METHOD PRIVATE RegisterWithDatatypes
VAR_INPUT
END_VAR
IF datatypes = 0 THEN
	RETURN;
END_IF

datatypes.OnEvent('OnDatatypeAdded',THIS^);
END_METHOD

METHOD PROTECTED CreateBundleNode : I_Node
VAR_INPUT
	NodeDatatype : I_StructuredDatatype;
END_VAR
VAR
	pAnyBundleNode : POINTER TO AnyBundleNode;
END_VAR
pAnyBundleNode := __NEW(AnyBundleNode(StructuredDatatype := NodeDatatype));
CreateBundleNode := pAnyBundleNode^;
END_METHOD

METHOD PROTECTED CreateDisplayNode : I_Node
VAR_INPUT
	NodeDatatype : I_Datatype;
END_VAR
VAR
	pAnyDisplayNode : POINTER TO AnyDisplayNode;
END_VAR
pAnyDisplayNode := __NEW(AnyDisplayNode(Datatype := NodeDatatype));
CreateDisplayNode := pAnyDisplayNode^;
END_METHOD

METHOD PROTECTED CreateLiteralNode : I_Node
VAR_INPUT
	NodeDatatype : I_Datatype;
END_VAR
VAR
	pAnyLiteralNode : POINTER TO AnyLiteralNode;
END_VAR
pAnyLiteralNode := __NEW(AnyLiteralNode(Datatype := NodeDatatype));
CreateLiteralNode := pAnyLiteralNode^;
END_METHOD

METHOD PROTECTED CreateUnbundleNode : I_Node
VAR_INPUT
	NodeDatatype : I_StructuredDatatype;
END_VAR
VAR
	pAnyUnbundleNode : POINTER TO AnyUnbundleNode;
END_VAR
pAnyUnbundleNode := __NEW(AnyUnbundleNode(StructuredDatatype := NodeDatatype));
CreateUnbundleNode := pAnyUnbundleNode^;
END_METHOD

METHOD PROTECTED RegisterBundleNodeOfType
VAR_INPUT
	NodeDatatype : I_StructuredDatatype;
END_VAR
VAR
	node : I_Node;
	path : T_MAXSTRING;
END_VAR
node := CreateBundleNode(NodeDatatype);
selfCreatedNodes.Push(node);
path := concat('Bundle/', NodeDatatype.Identifier);
nodeFactory.AddNodeAsPrototype(path,node);
END_METHOD

METHOD PROTECTED RegisterInterfaceDisplayNodeOfType
VAR_INPUT
	NodeDatatype : I_InterfaceDatatype;
END_VAR
VAR
	node : I_Node;
	path : T_MAXSTRING;
END_VAR
node := CreateDisplayNode(NodeDatatype);
selfCreatedNodes.Push(node);
path := concat('Display/', NodeDatatype.Identifier);
nodeFactory.AddNodeAsPrototype(path,node);
END_METHOD

METHOD PROTECTED RegisterInterfaceLiteralNodeOfType
VAR_INPUT
	NodeDatatype : I_InterfaceDatatype;
END_VAR
VAR
	node : I_Node;
	path : T_MAXSTRING;
END_VAR
node := CreateLiteralNode(NodeDatatype);
selfCreatedNodes.Push(node);
path := concat('Literal/', NodeDatatype.Identifier);
nodeFactory.AddNodeAsPrototype(path,node);
END_METHOD

METHOD PROTECTED RegisterPrimitiveDisplayNodeOfType
VAR_INPUT
	NodeDatatype : I_Datatype;
END_VAR
VAR
	node : I_Node;
	path : T_MAXSTRING;
END_VAR
node := CreateDisplayNode(NodeDatatype);
selfCreatedNodes.Push(node);
path := concat('Display/',NodeDatatype.TypeName);
nodeFactory.AddNodeAsPrototype(path,node);
END_METHOD

METHOD PROTECTED RegisterPrimitiveLiteralNodeOfType
VAR_INPUT
	NodeDatatype : I_Datatype;
END_VAR
VAR
	node : I_Node;
	path : T_MAXSTRING;
END_VAR
node := CreateLiteralNode(NodeDatatype);
selfCreatedNodes.Push(node);
path := concat('Literal/',NodeDatatype.TypeName);
nodeFactory.AddNodeAsPrototype(path,node);
END_METHOD

METHOD PROTECTED RegisterUdtDisplayNodeOfType
VAR_INPUT
	NodeDatatype : I_UserDefinedDatatype;
END_VAR
VAR
	node : I_Node;
	path : T_MAXSTRING;
END_VAR
node := CreateDisplayNode(NodeDatatype);
selfCreatedNodes.Push(node);
path := concat('Display/', NodeDatatype.Identifier);
nodeFactory.AddNodeAsPrototype(path,node);
END_METHOD

METHOD PROTECTED RegisterUdtLiteralNodeOfType
VAR_INPUT
	NodeDatatype : I_UserDefinedDatatype;
END_VAR
VAR
	node : I_Node;
	path : T_MAXSTRING;
END_VAR
node := CreateLiteralNode(NodeDatatype);
selfCreatedNodes.Push(node);
path := concat('Literal/', NodeDatatype.Identifier);
nodeFactory.AddNodeAsPrototype(path,node);
END_METHOD

METHOD PROTECTED RegisterUnbundleNodeOfType
VAR_INPUT
	NodeDatatype : I_StructuredDatatype;
END_VAR
VAR
	node : I_Node;
	path : T_MAXSTRING;
END_VAR
node := CreateUnbundleNode(NodeDatatype);
selfCreatedNodes.Push(node);
path := concat('Unbundle/', NodeDatatype.Identifier);
nodeFactory.AddNodeAsPrototype(path,node);
END_METHOD

METHOD PUBLIC HandleEvent
VAR_INPUT
	Event : I_Event;
END_VAR
VAR
	datatypeAddedEvent : I_DatatypeAddedEvent;
	aliasDatatypeAddedEvent : I_AliasDatatypeAddedEvent;
	enumDatatypeAddedEvent : I_EnumDatatypeAddedEvent;
	structuredDatatypeAddedEvent : I_StructuredDatatypeAddedEvent;
	interfaceDatatypeAddedEvent : I_InterfaceDatatypeAddedEvent;
END_VAR
IF __QUERYINTERFACE(event, datatypeAddedEvent) THEN
	RegisterPrimitiveLiteralNodeOfType(datatypeAddedEvent.Target);
	RegisterPrimitiveDisplayNodeOfType(datatypeAddedEvent.Target);
	RETURN;
END_IF

IF __QUERYINTERFACE(event, aliasDatatypeAddedEvent) THEN
	RegisterUdtLiteralNodeOfType(aliasDatatypeAddedEvent.Target);
	RegisterUdtDisplayNodeOfType(aliasDatatypeAddedEvent.Target);
	RETURN;
END_IF

IF __QUERYINTERFACE(event, enumDatatypeAddedEvent) THEN
	RegisterUdtLiteralNodeOfType(enumDatatypeAddedEvent.Target);
	RegisterUdtDisplayNodeOfType(enumDatatypeAddedEvent.Target);
	RETURN;
END_IF

IF __QUERYINTERFACE(event, interfaceDatatypeAddedEvent) THEN
	RegisterInterfaceLiteralNodeOfType(interfaceDatatypeAddedEvent.Target);
	RegisterInterfaceDisplayNodeOfType(interfaceDatatypeAddedEvent.Target);
	RETURN;
END_IF

IF __QUERYINTERFACE(event, structuredDatatypeAddedEvent) THEN
	RegisterUdtLiteralNodeOfType(structuredDatatypeAddedEvent.Target);
	RegisterUdtDisplayNodeOfType(structuredDatatypeAddedEvent.Target);
	RegisterBundleNodeOfType(structuredDatatypeAddedEvent.Target);
	RegisterUnbundleNodeOfType(structuredDatatypeAddedEvent.Target);
	RETURN;
END_IF
END_METHOD

END_FUNCTION_BLOCK

// Node/Bundle/AnyBundleNode
{attribute 'linkalways'} 
{attribute 'no_explicit_call' := 'This FB is a CLASS and must be accessed using methods or properties'}
{attribute 'enable_dynamic_creation'}
FUNCTION_BLOCK FINAL AnyBundleNode EXTENDS Node
VAR
	in : I_StructuredDatatype;
	out : I_StructuredDatatype;
	datatypeOperations : DatatypeOperations;
	selfMadeMembers : Stack;
END_VAR

METHOD FB_init : BOOL
VAR_INPUT
	bInitRetains : BOOL; // if TRUE, the retain variables are initialized (warm start / cold start)
	bInCopyCode : BOOL;  // if TRUE, the instance afterwards gets moved into the copy code (online change)
	StructuredDatatype : I_StructuredDatatype;
END_VAR
VAR
	enumerator : I_KeyValueForwardEnumerator;
	member : I_Datatype;
	memberAsBit : I_BitDatatype;
	memberAsBool : I_Datatype;
	_bool : pointer to _BOOL;
	memberClone : I_Datatype;
END_VAR
StructuredDatatype.Clone().TryResolveAsStructuredDatatype(out);
AddOutput('out', out);

StructuredDatatype.Clone().TryResolveAsStructuredDatatype(in);
enumerator := in.Members.GetMemberEnumerator();

WHILE enumerator.MoveNext() DO 
	IF enumerator.TryGet(member) THEN
		IF member.TryResolveAsBitDatatype(memberAsBit) THEN
			// if the element is a _bit then this needs to be treated differently (as you cannot simply memcpy
			// a bit, as it sits next to other data. Instead, a bool is added in it's place.	
			_bool := __NEW(_BOOL(InitialValue := memberAsBit.Value));
			datatypeOperations.AddWriteBoolToBitOperation(_bool^, memberAsBit);
			AddInput(enumerator.Key, _bool^);
			memberAsBool := _bool^;
			selfMadeMembers.Push(memberAsBool);
		ELSE
			// for all other datatypes,
			memberClone := member.Clone();
			datatypeOperations.AddMemoryCopyOperation(memberClone, member);
			AddInput(enumerator.key, memberClone);
			selfMadeMembers.Push(memberClone);
		END_IF
	END_IF
END_WHILE

enumerator.Dispose();
END_METHOD

METHOD FB_exit : BOOL
VAR_INPUT
	bInCopyCode : BOOL; // if TRUE, the exit method is called for exiting an instance that is copied afterwards (online change).
END_VAR
VAR
	member : I_Datatype;
END_VAR
IF bInCopyCode THEN
	RETURN;
END_IF

in.Dispose();
out.Dispose();
datatypeOperations.Clear();

WHILE selfMadeMembers.TryPop(member) DO
	IF member <> 0 THEN 
		member.dispose();
	END_IF
END_WHILE
END_METHOD

METHOD PUBLIC Clone : I_Node
VAR
	pNode : POINTER TO AnyBundleNode;
END_VAR
pNode := __NEW(AnyBundleNode(StructuredDatatype := in));
Clone := pNode^;
END_METHOD

METHOD PROTECTED OnExecute : HRESULT
VAR
END_VAR
datatypeOperations.Execute();
memcpy(out.Address, in.Address, in.Size);
END_METHOD

END_FUNCTION_BLOCK

// Node/Display/AnyDisplayNode
{attribute 'linkalways'} 
{attribute 'no_explicit_call' := 'This FB is a CLASS and must be accessed using methods or properties'}
{attribute 'enable_dynamic_creation'}
FUNCTION_BLOCK FINAL AnyDisplayNode EXTENDS Node
VAR
	in : I_Datatype;
	display : I_Datatype;
END_VAR

METHOD FB_init : BOOL
VAR_INPUT
	bInitRetains : BOOL; // if TRUE, the retain variables are initialized (warm start / cold start)
	bInCopyCode : BOOL;  // if TRUE, the instance afterwards gets moved into the copy code (online change)
	Datatype : I_Datatype;
END_VAR
THIS^.in := Datatype.Clone();
THIS^.display := Datatype.Clone();

AddInput('in', THIS^.in);
AddContent('display', THIS^.display);
END_METHOD

METHOD FB_exit : BOOL
VAR_INPUT
	bInCopyCode : BOOL; // if TRUE, the exit method is called for exiting an instance that is copied afterwards (online change).
END_VAR
IF bInCopyCode THEN
	RETURN;
END_IF

in.Dispose();
display.Dispose();
END_METHOD

METHOD PUBLIC Clone : I_Node
VAR
	pNode : POINTER TO AnyDisplayNode;
END_VAR
pNode := __NEW(AnyDisplayNode(Datatype := in));
Clone := pNode^;
END_METHOD

METHOD PROTECTED OnExecute : HRESULT
VAR
END_VAR
memcpy(display.Address, in.Address, in.Size);
END_METHOD

END_FUNCTION_BLOCK

// Node/Literal/AnyLiteralNode
{attribute 'linkalways'} 
{attribute 'no_explicit_call' := 'This FB is a CLASS and must be accessed using methods or properties'}
{attribute 'enable_dynamic_creation'}
FUNCTION_BLOCK FINAL AnyLiteralNode EXTENDS Node
VAR
	value : I_Datatype;
	out : I_Datatype;
END_VAR

METHOD FB_init : BOOL
VAR_INPUT
	bInitRetains : BOOL; // if TRUE, the retain variables are initialized (warm start / cold start)
	bInCopyCode : BOOL;  // if TRUE, the instance afterwards gets moved into the copy code (online change)
	Datatype : I_Datatype;
END_VAR
THIS^.value := Datatype.Clone();
THIS^.out := Datatype.Clone();

AddParameter('value', THIS^.value);
AddOutput('out', THIS^.out);
END_METHOD

METHOD FB_exit : BOOL
VAR_INPUT
	bInCopyCode : BOOL; // if TRUE, the exit method is called for exiting an instance that is copied afterwards (online change).
END_VAR
IF bInCopyCode THEN
	RETURN;
END_IF

value.Dispose();
out.Dispose();
END_METHOD

METHOD PUBLIC Clone : I_Node
VAR
	pNode : POINTER TO AnyLiteralNode;
END_VAR
pNode := __NEW(AnyLiteralNode(Datatype := value));
Clone := pNode^;
END_METHOD

METHOD PROTECTED OnExecute : HRESULT
VAR
END_VAR
memcpy(out.Address, value.Address, value.Size);
END_METHOD

END_FUNCTION_BLOCK

// Node/Unbundle/AnyUnbundleNode
{attribute 'linkalways'} 
{attribute 'no_explicit_call' := 'This FB is a CLASS and must be accessed using methods or properties'}
{attribute 'enable_dynamic_creation'}
FUNCTION_BLOCK FINAL AnyUnbundleNode EXTENDS Node
VAR
	in : I_StructuredDatatype;
	out : I_StructuredDatatype;
	datatypeOperations : DatatypeOperations;
	selfMadeMembers : Stack;
END_VAR

METHOD FB_init : BOOL
VAR_INPUT
	bInitRetains : BOOL; // if TRUE, the retain variables are initialized (warm start / cold start)
	bInCopyCode : BOOL;  // if TRUE, the instance afterwards gets moved into the copy code (online change)
	StructuredDatatype : I_StructuredDatatype;
END_VAR
VAR
	enumerator : I_KeyValueForwardEnumerator;
	member : I_Datatype;
	memberAsBit : I_BitDatatype;
	memberAsBool : I_Datatype;
	_bool : Pointer to _BOOL;
	memberClone : I_Datatype;
END_VAR
StructuredDatatype.Clone().TryResolveAsStructuredDatatype(in);
AddInput('in', in);

StructuredDatatype.Clone().TryResolveAsStructuredDatatype(out);
enumerator := out.Members.GetMemberEnumerator();

WHILE enumerator.MoveNext() DO 
	IF enumerator.TryGet(member) THEN
		IF member.TryResolveAsBitDatatype(memberAsBit) THEN
			// if the element is a _bit then this needs to be treated differently (as you cannot simply memcpy
			// a bit, as it sits next to other data. Instead, a bool is added in it's place.	
			_bool := __NEW(_BOOL(InitialValue := memberAsBit.Value));
			datatypeOperations.AddWriteBitToBoolOperation(memberAsBit, _bool^);
			AddOutput(enumerator.Key, _bool^);
			memberAsBool := _bool^;
			selfMadeMembers.Push(memberAsBool);
		ELSE
			// for all other datatypes,
			memberClone := member.Clone();
			datatypeOperations.AddMemoryCopyOperation(member, memberClone);
			AddOutput(enumerator.key, memberClone);
			selfMadeMembers.Push(memberClone);
		END_IF		
	END_IF
END_WHILE

enumerator.Dispose();
END_METHOD

METHOD FB_exit : BOOL
VAR_INPUT
	bInCopyCode : BOOL; // if TRUE, the exit method is called for exiting an instance that is copied afterwards (online change).
END_VAR
VAR
	member : I_Datatype;
END_VAR
IF bInCopyCode THEN
	RETURN;
END_IF

in.Dispose();
out.Dispose();
datatypeOperations.Clear();

WHILE selfMadeMembers.TryPop(member) DO
	IF member <> 0 THEN 
		member.dispose();
	END_IF
END_WHILE
END_METHOD

METHOD PUBLIC Clone : I_Node
VAR
	pNode : POINTER TO AnyUnbundleNode;
END_VAR
pNode := __NEW(AnyUnbundleNode(StructuredDatatype := in));
Clone := pNode^;
END_METHOD

METHOD PROTECTED OnExecute : HRESULT
VAR
END_VAR
memcpy(out.Address, in.Address, in.Size);
datatypeOperations.Execute();
END_METHOD

END_FUNCTION_BLOCK

// Graph/Base/Graph
{attribute 'linkalways'} 
{attribute 'no_explicit_call' := 'This FB is a CLASS and must be accessed using methods or properties'}
{attribute 'enable_dynamic_creation'}
FUNCTION_BLOCK Graph EXTENDS Disposable IMPLEMENTS I_Graph
VAR
	nodeFactory : I_NodeFactory;
	_uuid : T_MAXSTRING;	
	eventEmitter : EventEmitter;
	nodeHost : NodeHost(THIS^, eventEmitter);
	inputPortHost : InputPortHost(THIS^, eventEmitter);
	outputPortHost : OutputPortHost(THIS^, eventEmitter);
	parameterHost : ParameterHost(THIS^, eventEmitter);
	contentHost : ContentHost(THIS^, eventEmitter);
	alarmHost : AlarmHost(THIS^, eventEmitter);
	metadataHost : MetadataHost(THIS^, eventEmitter);
	extensionHost : ExtensionHost(THIS^,eventEmitter);
	selfCreatedNodes : Stack;
	
	deserializationFailedAlarm : DeserializationFailedAlarm(THIS^);
	deserializationFailedNodeNotSupportedAlarm : DeserializationFailedNodeNotSupportedAlarm(THIS^);
END_VAR

METHOD FB_init : BOOL
VAR_INPUT
	bInitRetains : BOOL; // if TRUE, the retain variables are initialized (warm start / cold start)
	bInCopyCode : BOOL;  // if TRUE, the instance afterwards gets moved into the copy code (online change)
	NodeFactory : I_NodeFactory;
END_VAR
THIS^.nodeFactory := NodeFactory;
END_METHOD

METHOD FB_exit : BOOL
VAR_INPUT
	bInCopyCode : BOOL; // if TRUE, the exit method is called for exiting an instance that is copied afterwards (online change).
END_VAR
IF bInCopyCode THEN
	RETURN;
END_IF

DisposeSelfCreatedNodes();
END_METHOD

METHOD PRIVATE DisposeSelfCreatedNodes : BOOL
VAR
	node : I_Node;
END_VAR
WHILE selfCreatedNodes.TryPop(node) DO
	nodeHost.RemoveNode(node);
	node.Dispose();
END_WHILE
END_METHOD

METHOD PUBLIC TryDeserializeLinks : BOOL
VAR_INPUT
	Deserializer : I_Deserializer;
	Feedback : I_DeserializerFeedback;
END_VAR
VAR
	linksDeserializer : I_Deserializer;
	linksEnumerator : I_DeserializerArrayForwardEnumerator;
	linkDeserializer : I_Deserializer;
	sourceNodeId : T_MAXSTRING;
	sourcePortName : T_MAXSTRING;
	destinationNodeId : T_MAXSTRING;
	destinationPortName : T_MAXSTRING;
	sourceNode : I_Node;
	sourcePort : I_OutputPort;
	destinationNode : I_Node;
	destinationPort : I_InputPort;
END_VAR
linksDeserializer := Deserializer.GetKeyArray('links');
linksEnumerator := linksDeserializer.GetArrayEnumerator();

WHILE linksEnumerator.MoveNext() DO
	
	linkDeserializer := linksEnumerator.Current.GetArray();
	
	IF NOT linkDeserializer.GetElementByIndex(1).TryGetString(sourceNodeId, Feedback) THEN
		DeserializationFailedAlarm.Raise('Missing source node id from link');
		linksEnumerator.Dispose();
		RETURN;
	END_IF
	
	IF NOT linkDeserializer.GetElementByIndex(2).TryGetString(sourcePortName, Feedback) THEN
		DeserializationFailedAlarm.Raise('Missing source port name from link');
		linksEnumerator.Dispose();
		RETURN;
	END_IF
	
	IF NOT linkDeserializer.GetElementByIndex(3).TryGetString(destinationNodeId, Feedback) THEN
		DeserializationFailedAlarm.Raise('Missing destination node id from link');
		linksEnumerator.Dispose();
		RETURN;
	END_IF
	
	IF NOT linkDeserializer.GetElementByIndex(4).TryGetString(destinationPortName, Feedback) THEN
		DeserializationFailedAlarm.Raise('Missing destination port name from link');
		linksEnumerator.Dispose();
		RETURN;
	END_IF
	
	IF NOT nodeHost.TryGetNodeById(sourceNodeId, sourceNode) THEN
		DeserializationFailedAlarm.Raise('Unable to get source node when creating link');
		linksEnumerator.Dispose();
		RETURN;
	END_IF
	
	IF NOT nodeHost.TryGetNodeById(destinationNodeId, destinationNode) THEN
		DeserializationFailedAlarm.Raise('Unable to get destination node when creating link');
		linksEnumerator.Dispose();
		RETURN;
	END_IF
	
	IF NOT sourceNode.OutputPorts.TryGetOutputPortByName(sourcePortName, sourcePort) THEN
		DeserializationFailedAlarm.Raise('Unable to get source port when creating link');
		linksEnumerator.Dispose();
		RETURN;
	END_IF
	
	IF NOT destinationNode.InputPorts.TryGetInputPortByName(destinationPortName, destinationPort) THEN
		DeserializationFailedAlarm.Raise('Unable to get destination port when creating link');
		linksEnumerator.Dispose();
		RETURN;
	END_IF
	
	IF NOT destinationPort.TryConnectTo(sourcePort) THEN
		DeserializationFailedAlarm.Raise('Unable to connect source to destination when creating link');
		linksEnumerator.Dispose();
		RETURN;
	END_IF
	
END_WHILE

TryDeserializeLinks := TRUE;
linksEnumerator.Dispose();
END_METHOD

METHOD PUBLIC TryDeserializeNodes : BOOL;
VAR_INPUT
	Deserializer : I_Deserializer;
	Feedback : I_DeserializerFeedback;
END_VAR
VAR
	nodeDeserializer : I_Deserializer;
	nodesEnumerator : I_DeserializerArrayForwardEnumerator;
	nodeType : T_MAXSTRING;
	pError : POINTER TO MissingNodePrototypeDeserializationError;
	node : I_Node;
END_VAR
nodeDeserializer := Deserializer.GetKeyArray('nodes');
nodesEnumerator := nodeDeserializer.GetArrayEnumerator();

WHILE nodesEnumerator.MoveNext() DO
	
	IF NOT nodesEnumerator.Current.TryGetKeyString('type',nodeType, Feedback) THEN
		RETURN;
	END_IF
	
	IF NOT nodeFactory.TryCreateNodeByType(nodeType, node) THEN
		pError := __NEW(MissingNodePrototypeDeserializationError(MissingType := nodeType));
		Feedback.LogError(pError^);
		DeserializationFailedNodeNotSupportedAlarm.Raise(nodeType);
		nodesEnumerator.Dispose();
		RETURN;
	END_IF
	
	selfCreatedNodes.Push(node);
	
	IF NOT node.TryDeserializeFrom(nodesEnumerator.Current, Feedback) THEN
		DeserializationFailedAlarm.Raise('Node failed to deserialize');
		nodesEnumerator.Dispose();
		RETURN;
	END_IF
	
	Nodes.AddNode(node);

END_WHILE

TryDeserializeNodes := TRUE;
nodesEnumerator.Dispose();
END_METHOD

METHOD PUBLIC Accept
VAR_INPUT
	Visitor : I_GraphVisitor;
END_VAR
Visitor.VisitGraph(THIS^);
END_METHOD

METHOD PUBLIC AddMetadata : I_HostMetadata
VAR_INPUT
	Name : T_MAXSTRING;
	Data : I_Datatype;
END_VAR
Metadatum.AddDataAsMetadata(Name, Data);
AddMetadata := THIS^;
END_METHOD

PROPERTY PUBLIC Alarms : I_Alarms
GET
Alarms := alarmHost;
END_GET
END_PROPERTY

PROPERTY PUBLIC Contents : I_Contents
GET
Contents := contentHost;
END_GET
END_PROPERTY

METHOD Execute
VAR_INPUT
END_VAR
nodeHost.Execute();
END_METHOD

PROPERTY PUBLIC Extensions : I_Extensions
GET
Extensions := extensionHost;
END_GET
END_PROPERTY

PROPERTY PUBLIC HasRaisedAlarm : BOOL
GET
HasRaisedAlarm := alarmHost.HasRaisedAlarm;
END_GET
END_PROPERTY

PROPERTY PUBLIC InputPorts : I_InputPorts
GET
InputPorts := inputPortHost;
END_GET
END_PROPERTY

PROPERTY PUBLIC Metadatum : I_Metadatum
GET
Metadatum := metadataHost;
END_GET
END_PROPERTY

PROPERTY PUBLIC Nodes : I_Nodes
GET
Nodes := nodeHost;
END_GET
END_PROPERTY

METHOD PUBLIC OffEvent
VAR_INPUT
	EventName : T_MaxString;
	EventHandler : I_EventHandler;
END_VAR
eventEmitter.OffEvent(EventName, EventHandler);
END_METHOD

METHOD PUBLIC OnceEvent
VAR_INPUT
	EventName : T_MaxString;
	EventHandler : I_EventHandler;
END_VAR
eventEmitter.OnceEvent(EventName, EventHandler);
END_METHOD

METHOD PUBLIC OnEvent
VAR_INPUT
	EventName : T_MaxString;
	EventHandler : I_EventHandler;
END_VAR
eventEmitter.OnEvent(EventName, EventHandler);
END_METHOD

PROPERTY PUBLIC OutputPorts : I_OutputPorts
GET
OutputPorts := outputPortHost;
END_GET
END_PROPERTY

PROPERTY PUBLIC Parameters : I_Parameters
GET
Parameters := parameterHost;
END_GET
END_PROPERTY

METHOD PUBLIC Reset
VAR_INPUT
END_VAR
_uuid := '';
DisposeSelfCreatedNodes();
END_METHOD

METHOD PUBLIC SerializeWith
VAR_INPUT
	Serializer : I_Serializer;
END_VAR
Serializer.StartObject();
Serializer.AddKeyString('uuid',_uuid);
inputPortHost.SerializeWith(Serializer);
outputPortHost.SerializeWith(Serializer);
parameterHost.SerializeWith(Serializer);
contentHost.SerializeWith(Serializer);
alarmHost.SerializeWith(Serializer);
extensionHost.SerializeWith(Serializer);
metadataHost.SerializeWith(Serializer);
nodeHost.SerializeWith(Serializer);
Serializer.EndObject();
END_METHOD

METHOD PUBLIC TryDeserializeFrom : BOOL
VAR_INPUT
	Deserializer : I_Deserializer;
	Feedback : I_DeserializerFeedback;
END_VAR
VAR
	receivedUuid : T_MAXSTRING;
END_VAR
DeserializationFailedNodeNotSupportedAlarm.Clear();
DeserializationFailedAlarm.Clear();

IF NOT parameterHost.TryDeserializeFrom(Deserializer, Feedback) THEN
	RETURN;
END_IF

IF NOT extensionHost.TryDeserializeFrom(Deserializer, Feedback) THEN
	RETURN;
END_IF

IF NOT Deserializer.TryGetKeyString('uuid', receivedUuid, Feedback) THEN
	RETURN;
END_IF

Reset();

IF NOT TryDeserializeNodes(Deserializer, Feedback) THEN 
	RETURN;
END_IF

IF NOT TryDeserializeLinks(Deserializer, Feedback) THEN
	RETURN;
END_IF

_uuid := receivedUuid;
TryDeserializeFrom := TRUE;
END_METHOD

PROPERTY PUBLIC Uuid : T_MAXSTRING
GET
Uuid := _uuid;
END_GET
END_PROPERTY

END_FUNCTION_BLOCK

// Node/Host/NodeHost
{attribute 'linkalways'} 
{attribute 'no_explicit_call' := 'This FB is a CLASS and must be accessed using methods or properties'}
{attribute 'enable_dynamic_creation'}
FUNCTION_BLOCK NodeHost IMPLEMENTS I_Nodes, I_Serializable
VAR
	hostParent : I_HostNodes;
	eventTarget : I_EventTarget;
	nodes : OrderedDictionary;
	nodesInExecutionOrder : LinkedList;
	executeEnumerator : I_ForwardEnumerator;
END_VAR

METHOD FB_init : BOOL
VAR_INPUT
	bInitRetains : BOOL; // if TRUE, the retain variables are initialized (warm start / cold start)
	bInCopyCode : BOOL;  // if TRUE, the instance afterwards gets moved into the copy code (online change)
	Parent : I_HostNodes;
	parentEventTarget : I_EventTarget;
END_VAR
hostParent := Parent;
eventTarget := parentEventTarget;
CreateExecuteEnumerator();
END_METHOD

METHOD FB_exit : BOOL
VAR_INPUT
	bInCopyCode : BOOL; // if TRUE, the exit method is called for exiting an instance that is copied afterwards (online change).
END_VAR
IF bInCopyCode THEN
	RETURN;
END_IF

DestroyExecuteEnumerator();
END_METHOD

METHOD PRIVATE CreateExecuteEnumerator
VAR_INPUT
END_VAR
IF executeEnumerator <> 0 THEN
	executeEnumerator.Dispose();
END_IF

executeEnumerator := nodesInExecutionOrder.GetEnumerator();
END_METHOD

METHOD PRIVATE DestroyExecuteEnumerator
VAR_INPUT
END_VAR
IF executeEnumerator <> 0 THEN
	executeEnumerator.Dispose();
END_IF
END_METHOD

METHOD PROTECTED EmitOnNodeAddedEvent
VAR_INPUT
	Node : I_Node;
END_VAR
VAR
	pNodeAddedEvent : POINTER TO NodeAddedEvent;
END_VAR
IF eventTarget = 0 THEN
	RETURN;
END_IF

pNodeAddedEvent := __NEW(NodeAddedEvent(Target := Node));
eventTarget.Emit('OnNodeAdded',pNodeAddedEvent^);
pNodeAddedEvent^.Dispose();
END_METHOD

METHOD PROTECTED UpdateExecutionOrder
VAR_INPUT
	Node : I_Node;
END_VAR
VAR
	currentPosition : I_LinkedListNode;
	currentNode : I_Node;
END_VAR
// is the list empty?
IF nodesInExecutionOrder.First = 0 THEN
	// if so, add our node first and jump out as done.
	nodesInExecutionOrder.AddFirst(Node);
	RETURN;
END_IF

// if not empty, then is our node higher priorty than the first in the list. 
nodesInExecutionOrder.First.TryGet(currentNode); 
IF currentNode.Order > Node.Order THEN
	// if yes, we are now first, jump out as done. 
	nodesInExecutionOrder.AddFirst(Node);
	RETURN;
END_IF

// here, the list has something in it, and we have less priority than the node in first place.

// get the last node in the list and remember this as "currentPosition" 
currentPosition := nodesInExecutionOrder.Last;

WHILE (TRUE) DO
	
	currentPosition.TryGet(currentNode); 
	// is the current position higer priority than our node?
	IF currentNode.Order <= Node.Order THEN
		// if so, then we go after, jump out as we are done. 
		nodesInExecutionOrder.AddAfter(currentPosition, Node);
		RETURN;
	END_IF
	
	// move one up the list towards the top and try again.
	currentPosition := currentPosition.Previous;

END_WHILE
END_METHOD

METHOD PUBLIC Accept
VAR_INPUT
	Visitor : I_NodeVisitor;
END_VAR
VAR
	enumerator : I_ForwardEnumerator;
	node : I_Node;
END_VAR
enumerator := nodes.GetEnumerator();

WHILE (enumerator.MoveNext()) DO
	
	IF enumerator.TryGet(node) THEN
		node.Accept(Visitor);
	END_IF

END_WHILE

enumerator.Dispose();
END_METHOD

METHOD PUBLIC AddNode
VAR_INPUT
	Node : I_Node;
END_VAR
nodes.AddOrUpdate(Node.id, Node);
UpdateExecutionOrder(Node);
EmitOnNodeAddedEvent(Node);
CreateExecuteEnumerator();
END_METHOD

METHOD PUBLIC Execute
VAR_INPUT
END_VAR
VAR
	node : I_Node;
END_VAR
executeEnumerator.Reset();

WHILE executeEnumerator.MoveNext() DO
	IF executeEnumerator.TryGet(node) THEN
		node.Execute();
	END_IF
END_WHILE
END_METHOD

PROPERTY PUBLIC HasNodes : BOOL
GET
HasNodes := NOT nodes.IsEmpty;
END_GET
END_PROPERTY

METHOD PUBLIC RemoveNode
VAR_INPUT
	Node : I_Node;
END_VAR
nodes.Remove(Node.Id);
nodesInExecutionOrder.Remove(Node);
CreateExecuteEnumerator();
END_METHOD

METHOD PUBLIC SerializeWith
VAR_INPUT
	Serializer : I_Serializer;
END_VAR
VAR
	enumerator : I_ForwardEnumerator;
	node : I_Node;
END_VAR
IF nodes.Count = 0 THEN
	RETURN;
END_IF

Serializer.AddKey('nodes');
Serializer.StartArray();

enumerator := nodes.GetEnumerator();

WHILE enumerator.MoveNext() DO
	IF enumerator.TryGet(node) THEN
		node.SerializeWith(Serializer);
	END_IF
END_WHILE

Serializer.EndArray();
enumerator.Dispose();
END_METHOD

METHOD PUBLIC TryDeserializeFrom : BOOL
VAR_INPUT
	Deserializer : I_Deserializer;
	Feedback : I_DeserializerFeedback;
END_VAR
VAR
	nodeDeserializer : I_Deserializer;
	nodesEnumerator : I_DeserializerArrayForwardEnumerator;
	nodeId : T_MAXSTRING;
	node : I_Node;
END_VAR
nodeDeserializer := Deserializer.GetKeyArray('nodes');
nodesEnumerator := nodeDeserializer.GetArrayEnumerator();

WHILE nodesEnumerator.MoveNext() DO
	
	IF NOT nodesEnumerator.Current.TryGetKeyString('id',nodeId, Feedback) THEN
		CONTINUE;
	END_IF
	
	IF NOT TryGetNodeById(nodeId, node)THEN
		CONTINUE;
	END_IF
	
	node.TryDeserializeFrom(nodesEnumerator.Current, Feedback);

END_WHILE

nodesEnumerator.Dispose();
END_METHOD

METHOD PUBLIC TryGetNodeById : BOOL
VAR_INPUT
	Id : T_MAXSTRING;
	Destination : REFERENCE TO I_Node;
END_VAR
VAR
	node : I_Node;
END_VAR
IF NOT nodes.TryGetValue(Id, node) THEN
	RETURN;
END_IF

Destination := node;
TryGetNodeById := TRUE;
END_METHOD

END_FUNCTION_BLOCK

// Node/Events/NodeAddedEvent
{attribute 'linkalways'} 
{attribute 'no_explicit_call' := 'This FB is a CLASS and must be accessed using methods or properties'}
{attribute 'enable_dynamic_creation'}
FUNCTION_BLOCK NodeAddedEvent EXTENDS Disposable IMPLEMENTS I_NodeAddedEvent
VAR
	_target : I_Node;
END_VAR

METHOD FB_init : BOOL
VAR_INPUT
	bInitRetains : BOOL; // if TRUE, the retain variables are initialized (warm start / cold start)
	bInCopyCode : BOOL;  // if TRUE, the instance afterwards gets moved into the copy code (online change)
	Target : I_Node;
END_VAR
This^._target := Target;
END_METHOD

PROPERTY PUBLIC Target : I_Node
GET
Target := _target;
END_GET
END_PROPERTY

END_FUNCTION_BLOCK

// Node/Events/I_NodeAddedEvent
INTERFACE I_NodeAddedEvent EXTENDS I_Event

PROPERTY PUBLIC Target : I_Node
GET
END_GET
END_PROPERTY

END_INTERFACE

// Errors/MissingNodePrototypeDeserializationError
{attribute 'linkalways'} 
{attribute 'no_explicit_call' := 'This FB is a CLASS and must be accessed using methods or properties'}
{attribute 'enable_dynamic_creation'}
FUNCTION_BLOCK MissingNodePrototypeDeserializationError EXTENDS Error
VAR
	nodeType : T_MAXSTRING;
END_VAR

METHOD FB_init : BOOL
VAR_INPUT
	bInitRetains : BOOL; // if TRUE, the retain variables are initialized (warm start / cold start)
	bInCopyCode : BOOL;  // if TRUE, the instance afterwards gets moved into the copy code (online change)
	MissingType : T_MAXSTRING;
END_VAR
 nodeType := MissingType;
END_METHOD

PROPERTY PUBLIC ErrorType : T_MAXSTRING
GET
ErrorType := 'MISSING_NODE_PROTOTYPE_DESERIALIZATION_ERROR';
END_GET
END_PROPERTY

PROPERTY PUBLIC Message : T_MAXSTRING
GET
Message := CONCAT('Deserialization Failed, Missing Node Prototype : ',nodeType);
END_GET
END_PROPERTY

END_FUNCTION_BLOCK

// Graph/Interfaces/I_Graphs
INTERFACE I_Graphs

METHOD PUBLIC Accept
VAR_INPUT
	visitor : I_GraphVisitor;
END_VAR
END_METHOD

METHOD PUBLIC AddGraph
VAR_INPUT
	Graph : I_Graph;
END_VAR
END_METHOD

METHOD PUBLIC DisposeAll
VAR_INPUT
END_VAR
END_METHOD

METHOD PUBLIC Execute
VAR_INPUT
END_VAR
END_METHOD

METHOD PUBLIC RemoveGraph
VAR_INPUT
	Graph : I_Graph;
END_VAR
END_METHOD

METHOD PUBLIC TryGetGraphByUuid : BOOL
VAR_INPUT
	Uuid : T_MAXSTRING;
	Destination : REFERENCE TO I_Graph;
END_VAR
END_METHOD

END_INTERFACE

// API/Visitors/GetStatusVisitor
{attribute 'linkalways'} 
{attribute 'no_explicit_call' := 'This FB is a CLASS and must be accessed using methods or properties'}
{attribute 'enable_dynamic_creation'}
FUNCTION_BLOCK GetStatusVisitor IMPLEMENTS I_GraphVisitor, I_NodeVisitor, I_ExtensionVisitor, I_ContentVisitor, I_AlarmVisitor
VAR
	serializer : I_Serializer;
END_VAR

METHOD PUBLIC Initialize
VAR_INPUT
	Serializer : I_Serializer;
END_VAR
THIS^.serializer := Serializer;
END_METHOD

METHOD VisitAlarm
VAR_INPUT
	VisitingAlarm : I_Alarm;
END_VAR
IF VisitingAlarm.Active THEN
	serializer.StartObject();
	serializer.AddKeyString('message',VisitingAlarm.Message);
	serializer.AddKeyString('reason',VisitingAlarm.Reason);
	serializer.EndObject();
END_IF
END_METHOD

METHOD VisitContent
VAR_INPUT
	VisitingContent : I_Content;
END_VAR
serializer.StartObject();

serializer.AddKeyString('name',VisitingContent.Name);
serializer.AddKeyObject('value',VisitingContent.Data);

serializer.EndObject();
END_METHOD

METHOD VisitExtension
VAR_INPUT
	VisitingExtension : I_Extension;
END_VAR
Serializer.StartObject();
Serializer.AddKeyString('name',VisitingExtension.Name);

IF VisitingExtension.Alarms.HasAlarms THEN
	serializer.addkey('alarms');
	serializer.StartArray();
	VisitingExtension.Alarms.Accept(THIS^);
	serializer.EndArray();
END_IF

IF VisitingExtension.Contents.HasContents THEN
	serializer.addkey('contents');
	serializer.StartArray();
	VisitingExtension.Contents.Accept(THIS^);
	serializer.EndArray();
END_IF

Serializer.EndObject();
END_METHOD

METHOD VisitGraph
VAR_INPUT
	VisitingGraph : I_Graph;
END_VAR
VAR
	includeInGetStatusVisitor : IncludeInGetStatusVisitor;
END_VAR
serializer.StartObject();

serializer.addKeyString('uuid',VisitingGraph.Uuid);

IF VisitingGraph.Alarms.HasRaisedAlarm THEN
	serializer.addkey('alarms');
	serializer.StartArray();
	VisitingGraph.Alarms.Accept(THIS^);
	serializer.EndArray();
END_IF

IF includeInGetStatusVisitor.CheckExtensions(VisitingGraph) THEN
	serializer.addkey('extensions');
	serializer.StartArray();
	VisitingGraph.Extensions.Accept(THIS^);
	serializer.EndArray();
END_IF

IF VisitingGraph.Contents.HasContents THEN
	serializer.addkey('contents');
	serializer.StartArray();
	VisitingGraph.Contents.Accept(THIS^);
	serializer.EndArray();
END_IF

IF VisitingGraph.Nodes.HasNodes THEN
	serializer.addkey('nodes');
	serializer.StartArray();
	VisitingGraph.Nodes.Accept(THIS^);
	serializer.EndArray();
END_IF

serializer.EndObject();
END_METHOD

METHOD VisitNode
VAR_INPUT
	VisitingNode : I_Node;
END_VAR
VAR
	includeInGetStatusVisitor : IncludeInGetStatusVisitor;
END_VAR
IF NOT includeInGetStatusVisitor.CheckNode(VisitingNode) THEN
	RETURN;
END_IF

serializer.StartObject();
serializer.addKeyString('id', VisitingNode.Id);

IF VisitingNode.Alarms.HasRaisedAlarm THEN
	serializer.addkey('alarms');
	serializer.StartArray();
	VisitingNode.Alarms.Accept(THIS^);
	serializer.EndArray();
END_IF

IF includeInGetStatusVisitor.CheckExtensions(VisitingNode) THEN
	serializer.addkey('extensions');
	serializer.StartArray();
	VisitingNode.Extensions.Accept(THIS^);
	serializer.EndArray();
END_IF

IF VisitingNode.Contents.HasContents THEN
	serializer.addkey('contents');
	serializer.StartArray();
	VisitingNode.Contents.Accept(THIS^);
	serializer.EndArray();
END_IF

serializer.EndObject();
END_METHOD

END_FUNCTION_BLOCK

// API/Visitors/IncludeInGetStatusVisitor
{attribute 'linkalways'} 
{attribute 'no_explicit_call' := 'This FB is a CLASS and must be accessed using methods or properties'}
{attribute 'enable_dynamic_creation'}
FUNCTION_BLOCK IncludeInGetStatusVisitor IMPLEMENTS I_NodeVisitor, I_ExtensionVisitor
VAR
	shouldInclude : BOOL;
END_VAR

METHOD PUBLIC CheckExtensions : BOOL;
VAR_INPUT
	ExtensionHost : I_HostExtensions;
END_VAR
shouldInclude := FALSE;
ExtensionHost.Extensions.Accept(THIS^);
CheckExtensions := shouldInclude;
END_METHOD

METHOD PUBLIC CheckNode : BOOL;
VAR_INPUT
	Node : I_Node;
END_VAR
shouldInclude := FALSE;
Node.Accept(THIS^);
CheckNode := shouldInclude;
END_METHOD

METHOD VisitExtension
VAR_INPUT
	VisitingExtension : I_Extension;
END_VAR
IF VisitingExtension.Contents.HasContents THEN
	shouldInclude := TRUE;
	RETURN;
END_IF

IF VisitingExtension.Alarms.HasRaisedAlarm THEN
	shouldInclude := TRUE;
	RETURN;
END_IF
END_METHOD

METHOD VisitNode
VAR_INPUT
	VisitingNode : I_Node;
END_VAR
IF VisitingNode.Contents.HasContents THEN
	shouldInclude := TRUE;
	RETURN;
END_IF

IF VisitingNode.Alarms.HasRaisedAlarm THEN
	shouldInclude := TRUE;
	RETURN;
END_IF

IF VisitingNode.Extensions.HasExtensions THEN
	VisitingNode.Extensions.Accept(THIS^);
END_IF
END_METHOD

END_FUNCTION_BLOCK

// API/Handlers/CreateGraphRpcHandler
{attribute 'linkalways'} 
{attribute 'no_explicit_call' := 'This FB is a CLASS and must be accessed using methods or properties'}
{attribute 'enable_dynamic_creation'}
FUNCTION_BLOCK CreateGraphRpcHandler IMPLEMENTS I_AsynchronousRpcHandler
VAR
	graphFramework : I_GraphFramework;
	graphs : I_Graphs;
	lastGraphUuid : T_MAXSTRING;
END_VAR

METHOD Handle
VAR_INPUT
	Parameters : I_Deserializer;
	Response : I_AsynchronousRpcResponse;
END_VAR
VAR
	graph : I_Graph;
	feedback : DeserializerFeedback;
	graphDeserializer : I_Deserializer;
	serializer : I_Serializer;
	getStatusVisitor : GetStatusVisitor;
END_VAR
IF graphs.TryGetGraphByUuid(lastGraphUuid,graph) THEN
	graphs.RemoveGraph(graph);
	graph.Dispose();
	lastGraphUuid := '';
END_IF

graph := graphFramework.Create();
graphDeserializer := Parameters.GetKeyObject('graph');

IF NOT graph.TryDeserializeFrom(graphDeserializer, feedback) THEN
	Response.RejectWithMessage(feedback.FirstError.Message);
	graph.Dispose();
	RETURN;
END_IF

lastGraphUuid := graph.Uuid;
graphs.AddGraph(graph);

serializer := Response.GetSerializer();
getStatusVisitor.Initialize(serializer);
getStatusVisitor.VisitGraph(graph);
Response.CompleteWithSerializer(serializer);
serializer.Dispose();
END_METHOD

METHOD PUBLIC Initialize
VAR_INPUT
	GraphFramework : I_GraphFramework;
	Graphs : I_Graphs;
END_VAR
THIS^.graphFramework := GraphFramework;
THIS^.graphs := Graphs;
END_METHOD

END_FUNCTION_BLOCK

// API/Handlers/GetBlueprintsRpcHandler
{attribute 'linkalways'} 
{attribute 'no_explicit_call' := 'This FB is a CLASS and must be accessed using methods or properties'}
{attribute 'enable_dynamic_creation'}
FUNCTION_BLOCK GetBlueprintsRpcHandler IMPLEMENTS I_AsynchronousRpcHandler
VAR
	nodeFactory : I_NodeFactory;
END_VAR

METHOD Handle
VAR_INPUT
	Parameters : I_Deserializer;
	Response : I_AsynchronousRpcResponse;
END_VAR
VAR
	visitor : GetBlueprintsVisitor;
	serializer : I_Serializer;
END_VAR
IF nodeFactory = 0 THEN
	Response.RejectWithMessage('GetBlueprintsRpcHandler has not been initialized with a valid nodeFactory object');
	RETURN;
END_IF

serializer := Response.GetSerializer();
visitor.Initialize(serializer);
nodeFactory.Accept(visitor);

Response.CompleteWithSerializer(serializer);
serializer.Dispose();
END_METHOD

METHOD PUBLIC Initialize
VAR_INPUT
	NodeFactory : I_NodeFactory;
END_VAR
this^.nodeFactory := NodeFactory;
END_METHOD

END_FUNCTION_BLOCK

// API/Visitors/GetBlueprintsVisitor
{attribute 'linkalways'} 
{attribute 'no_explicit_call' := 'This FB is a CLASS and must be accessed using methods or properties'}
{attribute 'enable_dynamic_creation'}
FUNCTION_BLOCK GetBlueprintsVisitor IMPLEMENTS I_NodeFactoryVisitor, I_NodePrototypeVisitor, I_NodeVisitor, I_ExtensionVisitor, I_InputPortVisitor, I_OutputPortVisitor, I_MetadataVisitor, I_ContentVisitor, I_ParameterVisitor, I_AlarmVisitor
VAR
	serializer : I_Serializer;
END_VAR

METHOD PUBLIC Initialize
VAR_INPUT
	Serializer : I_Serializer;
END_VAR
THIS^.serializer := Serializer;
END_METHOD

METHOD VisitAlarm
VAR_INPUT
	VisitingAlarm : I_Alarm;
END_VAR
serializer.AddString(VisitingAlarm.Message);
END_METHOD

METHOD VisitContent
VAR_INPUT
	VisitingContent : I_Content;
END_VAR
serializer.StartObject();

serializer.AddKeyString('name',VisitingContent.Name);
serializer.Addkey('datatype');
VisitingContent.Data.SerializeTypeWith(serializer);

IF VisitingContent.Metadatum.HasMetadata THEN
	serializer.addkey('metadata');
	serializer.StartArray();
	VisitingContent.Metadatum.Accept(THIS^);
	serializer.EndArray();
END_IF

serializer.EndObject();
END_METHOD

METHOD VisitExtension
VAR_INPUT
	VisitingExtension : I_Extension;
END_VAR
Serializer.StartObject();
Serializer.AddKeyString('name',VisitingExtension.Name);

IF VisitingExtension.Metadatum.HasMetadata THEN
	serializer.addkey('metadata');
	serializer.StartArray();
	VisitingExtension.Metadatum.Accept(THIS^);
	serializer.EndArray();
END_IF

IF VisitingExtension.Alarms.HasAlarms THEN
	serializer.addkey('alarms');
	serializer.StartArray();
	VisitingExtension.Alarms.Accept(THIS^);
	serializer.EndArray();
END_IF

IF VisitingExtension.InputPorts.HasInputPorts THEN
	serializer.addkey('inputPorts');
	serializer.StartArray();
	VisitingExtension.InputPorts.Accept(THIS^);
	serializer.EndArray();
END_IF

IF VisitingExtension.OutputPorts.HasOutputPorts THEN
	serializer.addkey('outputPorts');
	serializer.StartArray();
	VisitingExtension.OutputPorts.Accept(THIS^);
	serializer.EndArray();
END_IF

IF VisitingExtension.Parameters.HasParameters THEN
	serializer.addkey('parameters');
	serializer.StartArray();
	VisitingExtension.Parameters.Accept(THIS^);
	serializer.EndArray();
END_IF

IF VisitingExtension.Contents.HasContents THEN
	serializer.addkey('contents');
	serializer.StartArray();
	VisitingExtension.Contents.Accept(THIS^);
	serializer.EndArray();
END_IF

Serializer.EndObject();
END_METHOD

METHOD VisitInputPort
VAR_INPUT
	VisitingInputPort : I_InputPort;
END_VAR
serializer.StartObject();

serializer.AddKeyString('name',VisitingInputPort.Name);
serializer.Addkey('datatype');
VisitingInputPort.Data.SerializeTypeWith(serializer);

IF VisitingInputPort.Metadatum.HasMetadata THEN
	serializer.addkey('metadata');
	serializer.StartArray();
	VisitingInputPort.Metadatum.Accept(THIS^);
	serializer.EndArray();
END_IF

serializer.EndObject();
END_METHOD

METHOD VisitMetadatum
VAR_INPUT
	VisitingMetadatum : I_Metadata;
END_VAR
serializer.StartObject();
serializer.AddKeyString('name',VisitingMetadatum.Name);
serializer.AddkeyObject('value',VisitingMetadatum.Data);
serializer.EndObject();
END_METHOD

METHOD VisitNode
VAR_INPUT
	VisitingNode : I_Node;
END_VAR
serializer.StartObject();

IF VisitingNode.Metadatum.HasMetadata THEN
	serializer.addkey('metadata');
	serializer.StartArray();
	VisitingNode.Metadatum.Accept(THIS^);
	serializer.EndArray();
END_IF

IF VisitingNode.Alarms.HasAlarms THEN
	serializer.addkey('alarms');
	serializer.StartArray();
	VisitingNode.Alarms.Accept(THIS^);
	serializer.EndArray();
END_IF

IF VisitingNode.Extensions.HasExtensions THEN
	serializer.addkey('extensions');
	serializer.StartArray();
	VisitingNode.Extensions.Accept(THIS^);
	serializer.EndArray();
END_IF

IF VisitingNode.InputPorts.HasInputPorts THEN
	serializer.addkey('inputPorts');
	serializer.StartArray();
	VisitingNode.InputPorts.Accept(THIS^);
	serializer.EndArray();
END_IF

IF VisitingNode.OutputPorts.HasOutputPorts THEN
	serializer.addkey('outputPorts');
	serializer.StartArray();
	VisitingNode.OutputPorts.Accept(THIS^);
	serializer.EndArray();
END_IF

IF VisitingNode.Parameters.HasParameters THEN
	serializer.addkey('parameters');
	serializer.StartArray();
	VisitingNode.Parameters.Accept(THIS^);
	serializer.EndArray();
END_IF

IF VisitingNode.Contents.HasContents THEN
	serializer.addkey('contents');
	serializer.StartArray();
	VisitingNode.Contents.Accept(THIS^);
	serializer.EndArray();
END_IF

serializer.EndObject();
END_METHOD

METHOD VisitNodeFactory
VAR_INPUT
	VisitingNodeFactory : I_NodeFactory;
END_VAR
serializer.StartObject();
serializer.AddKey('blueprints');
serializer.StartArray();
VisitingNodeFactory.NodePrototypes.Accept(THIS^);
serializer.EndArray();
serializer.EndObject();
END_METHOD

METHOD VisitNodePrototype
VAR_INPUT
	VisitingPrototype : I_NodePrototype;
END_VAR
serializer.StartObject();
serializer.AddKeyString('path',VisitingPrototype.Path);
serializer.AddKey('node');
VisitingPrototype.Node.Accept(THIS^);
serializer.EndObject();
END_METHOD

METHOD VisitOutputPort
VAR_INPUT
	VisitingOutputPort : I_OutputPort;
END_VAR
serializer.StartObject();

serializer.AddKeyString('name',VisitingOutputPort.Name);
serializer.Addkey('datatype');
VisitingOutputPort.Data.SerializeTypeWith(serializer);

IF VisitingOutputPort.Metadatum.HasMetadata THEN
	serializer.addkey('metadata');
	serializer.StartArray();
	VisitingOutputPort.Metadatum.Accept(THIS^);
	serializer.EndArray();
END_IF

serializer.EndObject();
END_METHOD

METHOD VisitParameter
VAR_INPUT
	VisitingProperty : I_Parameter;
END_VAR
serializer.StartObject();

serializer.AddKeyString('name',VisitingProperty.Name);
serializer.Addkey('datatype');
VisitingProperty.Data.SerializeTypeWith(serializer);
serializer.Addkey('defaultValue');
VisitingProperty.Data.SerializeWith(serializer);

IF VisitingProperty.Metadatum.HasMetadata THEN
	serializer.addkey('metadata');
	serializer.StartArray();
	VisitingProperty.Metadatum.Accept(THIS^);
	serializer.EndArray();
END_IF

Serializer.EndObject();
END_METHOD

END_FUNCTION_BLOCK

// API/Handlers/GetContentValueHandler
{attribute 'linkalways'} 
{attribute 'no_explicit_call' := 'This FB is a CLASS and must be accessed using methods or properties'}
{attribute 'enable_dynamic_creation'}
FUNCTION_BLOCK GetContentValueHandler IMPLEMENTS I_AsynchronousRpcHandler
VAR
	graphs : I_Graphs;
END_VAR

METHOD Handle
VAR_INPUT
	Parameters : I_Deserializer;
	Response : I_AsynchronousRpcResponse;
END_VAR
VAR
	graphUuid : T_MAXSTRING;
	nodeId : T_MAXSTRING;
	contentName : T_MAXSTRING;
	visitor : RetrieveNodeContentValue;
	serializer : I_Serializer;
	feedback : DeserializerFeedback;
END_VAR
IF NOT Parameters.TryGetKeyString('graphUuid', graphUuid, feedback) THEN
	Response.RejectWithMessage(feedback.FirstError.Message);
	RETURN;
END_IF

IF NOT Parameters.TryGetKeyString('nodeId', nodeId, feedback) THEN
	Response.RejectWithMessage(feedback.FirstError.Message);
	RETURN;
END_IF

IF NOT Parameters.TryGetKeyString('contentName', contentName, feedback) THEN
	Response.RejectWithMessage(feedback.FirstError.Message);
	RETURN;
END_IF

serializer := Response.GetSerializer();
visitor.Initialize(graphUuid, nodeId, contentName, serializer);
graphs.Accept(visitor);

IF visitor.Error THEN
	Response.RejectWithMessage(visitor.ErrorMessage);
	serializer.Dispose();
	RETURN;
END_IF

IF NOT visitor.Done THEN
	Response.RejectWithMessage('Invalid graphUuid');
	serializer.Dispose();
	RETURN;
END_IF

Response.CompleteWithSerializer(serializer);
serializer.Dispose();
END_METHOD

METHOD PUBLIC Initialize
VAR_INPUT
	Graphs : I_Graphs;
END_VAR
this^.graphs := Graphs;
END_METHOD

END_FUNCTION_BLOCK

// API/Visitors/RetrieveNodeContentValue
{attribute 'linkalways'} 
{attribute 'no_explicit_call' := 'This FB is a CLASS and must be accessed using methods or properties'}
{attribute 'enable_dynamic_creation'}
FUNCTION_BLOCK RetrieveNodeContentValue IMPLEMENTS I_GraphVisitor, I_NodeVisitor, I_ContentVisitor
VAR
	graphUuid : T_MAXSTRING;
	nodeId : T_MAXSTRING;
	contentName : T_MAXSTRING;
	serializer : I_Serializer;
	_done : BOOL;
	_error : BOOL;
	_errorMessage : T_MAXSTRING;
END_VAR

METHOD PRIVATE LogInvalidContentNameError
VAR_INPUT
END_VAR
_errorMessage := 'Invalid Content Name';
_error := TRUE;
END_METHOD

METHOD PRIVATE LogInvalidNodeIdError
VAR_INPUT
END_VAR
_errorMessage := 'Invalid Node Id';
_error := TRUE;
END_METHOD

METHOD PRIVATE Reset
VAR_INPUT
END_VAR
_done := FALSE;
_errorMessage := '';
_error := FALSE;
END_METHOD

PROPERTY PUBLIC Done : BOOL
GET
Done := _done;
END_GET
END_PROPERTY

PROPERTY PUBLIC Error : BOOL
GET
Error := _error;
END_GET
END_PROPERTY

PROPERTY PUBLIC ErrorMessage : T_MAXSTRING
GET
ErrorMessage := _errorMessage;
END_GET
END_PROPERTY

METHOD PUBLIC Initialize
VAR_INPUT
	GraphUuid : T_MAXSTRING;
	NodeId : T_MAXSTRING;
	ContentName : T_MAXSTRING;
	Serializer : I_Serializer;
END_VAR
THIS^.graphUuid := GraphUuid;
THIS^.nodeId := NodeId;
THIS^.contentName := ContentName;
THIS^.serializer := Serializer;
END_METHOD

METHOD VisitContent
VAR_INPUT
	VisitingContent : I_Content;
END_VAR
VisitingContent.SerializeWith(serializer);
END_METHOD

METHOD VisitGraph
VAR_INPUT
	VisitingGraph : I_Graph;
END_VAR
VAR
	node : I_Node;
END_VAR
Reset();

IF NOT (VisitingGraph.Uuid = graphUuid) THEN
	RETURN;
END_IF

IF NOT VisitingGraph.Nodes.TryGetNodeById(nodeId, node) THEN
	LogInvalidNodeIdError();
	RETURN;
END_IF

node.Accept(THIS^);
END_METHOD

METHOD VisitNode
VAR_INPUT
	VisitingNode : I_Node;
END_VAR
VAR
	content : I_Content;
END_VAR
IF NOT VisitingNode.Contents.TryGetContentByName(contentName, content) THEN
	LogInvalidContentNameError();
	RETURN;
END_IF

content.Accept(THIS^);
END_METHOD

END_FUNCTION_BLOCK

// API/Handlers/GetStatusRpcHandler
{attribute 'linkalways'} 
{attribute 'no_explicit_call' := 'This FB is a CLASS and must be accessed using methods or properties'}
{attribute 'enable_dynamic_creation'}
FUNCTION_BLOCK GetStatusRpcHandler IMPLEMENTS I_AsynchronousRpcHandler
VAR
	graphs : I_Graphs;
END_VAR

METHOD Handle
VAR_INPUT
	Parameters : I_Deserializer;
	Response : I_AsynchronousRpcResponse;
END_VAR
VAR
	graphUuid : T_MAXSTRING;
	graph : I_Graph;
	feedback : DeserializerFeedback;
	serializer : I_Serializer;
	getStatusVisitor : GetStatusVisitor;
END_VAR
IF NOT Parameters.TryGetKeyString('graphUuid', graphUuid, feedback) THEN
	Response.RejectWithMessage(feedback.FirstError.Message);
	RETURN;
END_IF

IF NOT graphs.TryGetGraphByUuid(graphUuid,graph) THEN
	Response.RejectWithMessage(concat('Unknown UUID : ',graphUuid));
	RETURN;
END_IF

serializer := Response.GetSerializer();
getStatusVisitor.Initialize(serializer);
getStatusVisitor.VisitGraph(graph);
Response.CompleteWithSerializer(serializer);
serializer.Dispose();
END_METHOD

METHOD PUBLIC Initialize
VAR_INPUT
	Graphs : I_Graphs;
END_VAR
THIS^.graphs := Graphs;
END_METHOD

END_FUNCTION_BLOCK

// API/Handlers/UpdateParameterValueHandler
{attribute 'linkalways'} 
{attribute 'no_explicit_call' := 'This FB is a CLASS and must be accessed using methods or properties'}
{attribute 'enable_dynamic_creation'}
FUNCTION_BLOCK UpdateParameterValueHandler IMPLEMENTS I_AsynchronousRpcHandler
VAR
	graphs : I_Graphs;
END_VAR

METHOD Handle
VAR_INPUT
	Parameters : I_Deserializer;
	Response : I_AsynchronousRpcResponse;
END_VAR
VAR
	graphUuid : T_MAXSTRING;
	graph : I_Graph;
	nodeId : T_MAXSTRING;
	node : I_Node;
	parameterName : T_MAXSTRING;
	parameter : I_Parameter;
	visitor : RetrieveNodeContentValue;
	serializer : I_Serializer;
	feedback : DeserializerFeedback;
END_VAR
IF NOT Parameters.TryGetKeyString('graphUuid', graphUuid, feedback) THEN
	Response.RejectWithMessage(feedback.FirstError.Message);
	RETURN;
END_IF

IF NOT graphs.TryGetGraphByUuid(graphUuid, graph) THEN
	Response.RejectWithMessage('Invalid or missing graphUuid');
	RETURN;
END_IF

IF NOT Parameters.TryGetKeyString('nodeId', nodeId, feedback) THEN
	Response.RejectWithMessage(feedback.FirstError.Message);
	RETURN;
END_IF

IF NOT graph.Nodes.TryGetNodeById(nodeId, node) THEN
	Response.RejectWithMessage('Invalid or missing nodeId');
	RETURN;
END_IF

IF NOT Parameters.TryGetKeyString('parameterName', parameterName, feedback) THEN
	Response.RejectWithMessage(feedback.FirstError.Message);
	RETURN;
END_IF

IF NOT node.Parameters.TryGetParameterByName(parameterName, parameter) THEN
	Response.RejectWithMessage('Invalid or missing parameterName');
	RETURN;
END_IF

IF NOT Parameters.TryDeserializeKeyToObject ('parameterValue', parameter, feedback) THEN
	Response.RejectWithMessage(feedback.FirstError.Message);
	RETURN;
END_IF

Response.CompleteWithString('done');
END_METHOD

METHOD PUBLIC Initialize
VAR_INPUT
	Graphs : I_Graphs;
END_VAR
this^.graphs := Graphs;
END_METHOD

END_FUNCTION_BLOCK

// API/GraphFrameworkApi
{attribute 'linkalways'} 
{attribute 'no_explicit_call' := 'This FB is a CLASS and must be accessed using methods or properties'}
{attribute 'enable_dynamic_creation'}
FUNCTION_BLOCK GraphFrameworkApi IMPLEMENTS I_RpcApi, I_HostGraphs, I_EventEmitter
VAR
	graphFramework : I_GraphFramework;
	eventEmitter : EventEmitter;
	graphHost : GraphHost(THIS^, eventEmitter);
	createGraphRpcHandler : CreateGraphRpcHandler;
	createGraphMultiUserRpcHandler : CreateGraphMultiUserRpcHandler;
	getStatusRpcHandler : GetStatusRpcHandler;
	getBlueprintsRpcHandler : GetBlueprintsRpcHandler;
	getContentValueHandler : GetContentValueHandler;
	updateParameterValueHandler : UpdateParameterValueHandler;
END_VAR

METHOD FB_init : BOOL
VAR_INPUT
	bInitRetains : BOOL; // if TRUE, the retain variables are initialized (warm start / cold start)
	bInCopyCode : BOOL;  // if TRUE, the instance afterwards gets moved into the copy code (online change)
	GraphFramework : I_GraphFramework;
END_VAR
THIS^.graphFramework := GraphFramework;

getBlueprintsRpcHandler.Initialize(GraphFramework.NodeFactory);
getStatusRpcHandler.Initialize(graphHost);
createGraphRpcHandler.Initialize(GraphFramework, graphHost);
createGraphMultiUserRpcHandler.Initialize(GraphFramework, graphHost);
getContentValueHandler.Initialize(graphHost);
updateParameterValueHandler.Initialize(graphHost);
END_METHOD

METHOD FB_exit : BOOL
VAR_INPUT
	bInCopyCode : BOOL; // if TRUE, the exit method is called for exiting an instance that is copied afterwards (online change).
END_VAR
IF bInCopyCode THEN
	RETURN;
END_IF

graphs.DisposeAll();
END_METHOD

METHOD PUBLIC CyclicCall
VAR_INPUT
END_VAR
graphHost.Execute();
END_METHOD

PROPERTY PUBLIC Graphs : I_Graphs
GET
Graphs := graphHost;
END_GET
END_PROPERTY

METHOD PUBLIC OffEvent
VAR_INPUT
	EventName : T_MaxString;
	EventHandler : I_EventHandler;
END_VAR
eventEmitter.OffEvent(EventName, EventHandler);
END_METHOD

METHOD PUBLIC OnceEvent
VAR_INPUT
	EventName : T_MaxString;
	EventHandler : I_EventHandler;
END_VAR
eventEmitter.OnceEvent(EventName, EventHandler);
END_METHOD

METHOD PUBLIC OnEvent
VAR_INPUT
	EventName : T_MaxString;
	EventHandler : I_EventHandler;
END_VAR
eventEmitter.OnEvent(EventName, EventHandler);
END_METHOD

METHOD RegisterAsynchronousRpcHandlersWith
VAR_INPUT
	Host : I_HostAsynchronousRpcHandlers;
END_VAR
Host.RegisterHandler('CreateGraph',createGraphRpcHandler);
Host.RegisterHandler('CreateGraphMultiUser',createGraphMultiUserRpcHandler);
Host.RegisterHandler('GetStatus',getStatusRpcHandler);
Host.RegisterHandler('GetBlueprints',getBlueprintsRpcHandler);
Host.RegisterHandler('GetContentValue',getContentValueHandler);
Host.RegisterHandler('UpdateParameterValue',updateParameterValueHandler);
END_METHOD

METHOD RegisterSynchronousRpcHandlersWith
VAR_INPUT
	Host : I_HostSynchronousRpcHandlers;
END_VAR
// no implementation
END_METHOD

END_FUNCTION_BLOCK

// Graph/Interfaces/I_HostGraphs
INTERFACE I_HostGraphs

PROPERTY Graphs : I_Graphs
GET
END_GET
END_PROPERTY

END_INTERFACE

// Graph/Host/GraphHost
{attribute 'linkalways'} 
{attribute 'no_explicit_call' := 'This FB is a CLASS and must be accessed using methods or properties'}
{attribute 'enable_dynamic_creation'}
FUNCTION_BLOCK GraphHost IMPLEMENTS I_Graphs, I_Serializable
VAR
	hostParent : I_HostGraphs;
	eventTarget : I_EventTarget;
	graphs : OrderedDictionary;	
END_VAR

METHOD FB_init : BOOL
VAR_INPUT
	bInitRetains : BOOL; // if TRUE, the retain variables are initialized (warm start / cold start)
	bInCopyCode : BOOL;  // if TRUE, the instance afterwards gets moved into the copy code (online change)
	Parent : I_HostGraphs;
	ParentEventTarget : I_EventTarget;
END_VAR
hostParent := Parent;
eventTarget := parentEventTarget;
END_METHOD

METHOD PROTECTED EmitOnGraphAddedEvent
VAR_INPUT
	Graph : I_Graph;
END_VAR
VAR
	pGraphAddedEvent : POINTER TO GraphAddedEvent;
END_VAR
IF eventTarget = 0 THEN
	RETURN;
END_IF

pGraphAddedEvent := __NEW(GraphAddedEvent(Target := Graph));
eventTarget.Emit('OnGraphAdded',pGraphAddedEvent^);
pGraphAddedEvent^.Dispose();
END_METHOD

METHOD PUBLIC Accept
VAR_INPUT
	visitor : I_GraphVisitor;
END_VAR
VAR
	enumerator : I_ForwardEnumerator;
	graph : I_Graph;
END_VAR
enumerator := graphs.GetEnumerator();

WHILE (enumerator.MoveNext()) DO
	
	IF enumerator.TryGet(graph) THEN
		graph.Accept(Visitor);
	END_IF

END_WHILE

enumerator.Dispose();
END_METHOD

METHOD PUBLIC AddGraph
VAR_INPUT
	Graph : I_Graph;
END_VAR
graphs.AddOrUpdate(Graph.Uuid, Graph);
EmitOnGraphAddedEvent(Graph);
END_METHOD

METHOD PUBLIC DisposeAll
VAR_INPUT
END_VAR
VAR
	enumerator : I_ForwardEnumerator;
	graph : I_Graph;
END_VAR
enumerator := graphs.GetEnumerator();

WHILE enumerator.MoveNext() DO
	IF enumerator.TryGet(graph) THEN
		graph.Dispose();
	END_IF
END_WHILE

graphs.Clear();

enumerator.Dispose();
END_METHOD

METHOD PUBLIC Execute
VAR_INPUT
END_VAR
VAR
	enumerator : I_ForwardEnumerator;
	graph : I_Graph;
END_VAR
enumerator := graphs.GetEnumerator();

WHILE enumerator.MoveNext() DO
	IF enumerator.TryGet(graph) THEN
		graph.Execute();
	END_IF
END_WHILE

enumerator.Dispose();
END_METHOD

METHOD PUBLIC RemoveGraph
VAR_INPUT
	Graph : I_Graph;
END_VAR
graphs.Remove(Graph.Uuid);
END_METHOD

METHOD PUBLIC SerializeWith
VAR_INPUT
	Serializer : I_Serializer;
END_VAR
VAR
	enumerator : I_ForwardEnumerator;
	graph : I_Graph;
END_VAR
IF graphs.Count = 0 THEN
	RETURN;
END_IF

Serializer.AddKey('graphs');
Serializer.StartArray();

enumerator := graphs.GetEnumerator();

WHILE enumerator.MoveNext() DO
	IF enumerator.TryGet(graph) THEN
		graph.SerializeWith(Serializer);
	END_IF
END_WHILE

Serializer.EndArray();
enumerator.Dispose();
END_METHOD

METHOD PUBLIC TryGetGraphByUuid : BOOL
VAR_INPUT
	Uuid : T_MAXSTRING;
	Destination : REFERENCE TO I_Graph;
END_VAR
VAR
	graph : I_Graph;
END_VAR
IF NOT graphs.TryGetValue(Uuid, graph) THEN
	RETURN;
END_IF

Destination := graph;
TryGetGraphByUuid := TRUE;
END_METHOD

END_FUNCTION_BLOCK

// Graph/Events/GraphAddedEvent
{attribute 'linkalways'} 
{attribute 'no_explicit_call' := 'This FB is a CLASS and must be accessed using methods or properties'}
{attribute 'enable_dynamic_creation'}
FUNCTION_BLOCK GraphAddedEvent EXTENDS Disposable IMPLEMENTS I_GraphAddedEvent
VAR
	_target : I_Graph;
END_VAR

METHOD FB_init : BOOL
VAR_INPUT
	bInitRetains : BOOL; // if TRUE, the retain variables are initialized (warm start / cold start)
	bInCopyCode : BOOL;  // if TRUE, the instance afterwards gets moved into the copy code (online change)
	Target : I_Graph;
END_VAR
This^._target := Target;
END_METHOD

PROPERTY PUBLIC Target : I_Graph
GET
Target := _target;
END_GET
END_PROPERTY

END_FUNCTION_BLOCK

// Graph/Events/I_GraphAddedEvent
INTERFACE I_GraphAddedEvent EXTENDS I_Event

PROPERTY PUBLIC Target : I_Graph
GET
END_GET
END_PROPERTY

END_INTERFACE

// Extensions/Namespace/ExtensionNamespace
{attribute 'linkalways'} 
{attribute 'no_explicit_call' := 'This FB is a CLASS and must be accessed using methods or properties'}
{attribute 'enable_dynamic_creation'}
FUNCTION_BLOCK ExtensionNamespace
VAR
	_extensionName : T_MAXSTRING;
	_targetName : T_MAXSTRING;
	_isExtensionPath : BOOL;
END_VAR

METHOD FB_init : BOOL
VAR_INPUT
	bInitRetains : BOOL; // if TRUE, the retain variables are initialized (warm start / cold start)
	bInCopyCode : BOOL;  // if TRUE, the instance afterwards gets moved into the copy code (online change)
	Path : T_MAXSTRING;
END_VAR
Initialize(Path);
END_METHOD

PROPERTY PUBLIC ExtensionName : T_MAXSTRING
GET
IF NOT _isExtensionPath THEN
	RETURN;
END_IF

ExtensionName := _extensionNAme;
END_GET
END_PROPERTY

METHOD PUBLIC Initialize
VAR_INPUT
	Path : T_MAXSTRING;
END_VAR
_isExtensionPath := FindAndSplitChar(
	sSeparatorChar := '.',  
	pSrcString := ADR(Path),                                  
	pLeftString := ADR(_extensionName),   
	nLeftSize := SIZEOF(_extensionName),                                  
	pRightString := ADR(_targetName), 
	nRightSize := SIZEOF(_targetName),                                
	bSearchFromRight := TRUE 
);
END_METHOD

PROPERTY PUBLIC IsExtensionPath : BOOL
GET
IsExtensionPath := _isExtensionPath;
END_GET
END_PROPERTY

PROPERTY PUBLIC TargetName : T_MAXSTRING
GET
IF NOT _isExtensionPath THEN
	RETURN;
END_IF

TargetName := _targetName;
END_GET
END_PROPERTY

END_FUNCTION_BLOCK

// Extensions/PreExecutionCheck/Alarms/PreExecutionCheckFailedAlarm
{attribute 'linkalways'} 
{attribute 'no_explicit_call' := 'This FB is a CLASS and must be accessed using methods or properties'}
{attribute 'enable_dynamic_creation'}
FUNCTION_BLOCK PUBLIC PreExecutionCheckFailedAlarm EXTENDS Alarm
VAR
	state : (CLEARED, RAISED);
	_reason : T_MAXSTRING;
END_VAR

PROPERTY Active : BOOL
GET
Active := state <> CLEARED;
END_GET
END_PROPERTY

METHOD PUBLIC Clear
_reason := '';
state := CLEARED;
END_METHOD

PROPERTY PUBLIC Message : T_MaxString
GET
Message := 'Pre-execution check failed';
END_GET
END_PROPERTY

METHOD PUBLIC Raise
VAR_INPUT
	Reason : T_MAXSTRING;
END_VAR
_reason := Reason;
state := RAISED;
END_METHOD

PROPERTY Reason : T_MaxString
GET
Reason := _reason;
END_GET
END_PROPERTY

END_FUNCTION_BLOCK

// Extensions/PreExecutionCheck/Checks/I_PreExecutionChecks
INTERFACE I_PreExecutionChecks

METHOD PUBLIC Fail
VAR_INPUT
	Message : T_MAXSTRING;
END_VAR
END_METHOD

PROPERTY PUBLIC Failed : BOOL
GET
END_GET
END_PROPERTY

METHOD PUBLIC IsFalse
VAR_INPUT
	Actual : BOOL;
	Message : T_MAXSTRING;
END_VAR
END_METHOD

METHOD PUBLIC IsTrue
VAR_INPUT
	Actual : BOOL;
	Message : T_MAXSTRING;
END_VAR
END_METHOD

END_INTERFACE

// Extensions/PreExecutionCheck/Checks/PreExecutionChecks
FUNCTION_BLOCK PreExecutionChecks IMPLEMENTS I_PreExecutionChecks
VAR
	hasFailed : BOOL;
	hasFailedReason : T_MAXSTRING;
END_VAR;

METHOD PUBLIC Fail
VAR_INPUT
	Message : T_MAXSTRING;
END_VAR
IF hasFailed THEN
	RETURN;
END_IF

hasFailed := TRUE;
hasFailedReason := Message;
END_METHOD

PROPERTY PUBLIC Failed : BOOL
GET
Failed := hasFailed;
END_GET
END_PROPERTY

METHOD PUBLIC IsFalse
VAR_INPUT
	Actual : BOOL;
	Message : T_MAXSTRING;
END_VAR
IF hasFailed THEN
	RETURN;
END_IF

IF NOT Actual THEN
	RETURN;
END_IF

hasFailed := TRUE;
hasFailedReason := Message;
END_METHOD

METHOD PUBLIC IsTrue
VAR_INPUT
	Actual : BOOL;
	Message : T_MAXSTRING;
END_VAR
IF hasFailed THEN
	RETURN;
END_IF

IF Actual THEN
	RETURN;
END_IF

hasFailed := TRUE;
hasFailedReason := Message;
END_METHOD

PROPERTY PUBLIC Passed : BOOL
GET
Passed := not hasFailed;
END_GET
END_PROPERTY

PROPERTY PUBLIC Reason : T_MAXSTRING
GET
Reason := hasFailedReason;
END_GET
END_PROPERTY

METHOD PUBLIC Reset
VAR_INPUT
END_VAR
hasFailed := FALSE;
hasFailedReason := '';
END_METHOD

END_FUNCTION_BLOCK

// Extensions/PreExecutionCheck/Interfaces/I_PreCheckedNode
INTERFACE I_PreCheckedNode EXTENDS I_Node

METHOD PreExecutionCheck
VAR_INPUT
	Check : I_PreExecutionChecks;
END_VAR
END_METHOD

END_INTERFACE

// Extensions/PreExecutionCheck/PreExecutionCheckExtension
FUNCTION_BLOCK PreExecutionCheckExtension EXTENDS Extension IMPLEMENTS I_EventHandler
VAR
	parentAsPreCheckedNode : I_PreCheckedNode;
	preExecutionCheckFailedAlarm : PreExecutionCheckFailedAlarm(THIS^);
	enable : _BOOL(TRUE);
END_VAR

METHOD FB_init : BOOL
VAR_INPUT
	bInitRetains : BOOL; // if TRUE, the retain variables are initialized (warm start / cold start)
	bInCopyCode : BOOL;  // if TRUE, the instance afterwards gets moved into the copy code (online change)
	Name : T_MAXSTRING;
	Parent : I_HostExtensions;
END_VAR
AddParameter('enable', enable);

IF NOT __QUERYINTERFACE(Parent, parentAsPreCheckedNode) THEN
	RETURN;
END_IF

RegisterForPreExecuteEvent();
END_METHOD

METHOD FB_exit : BOOL
VAR_INPUT
	bInCopyCode : BOOL; // if TRUE, the exit method is called for exiting an instance that is copied afterwards (online change).
END_VAR
IF bInCopyCode THEN
	RETURN;
END_IF

DeregisterForPreExecuteEvent();
END_METHOD

METHOD PRIVATE DeregisterForPreExecuteEvent
VAR_INPUT
END_VAR
IF parentAsPreCheckedNode = 0 THEN
	RETURN;
END_IF

parentAsPreCheckedNode.OffEvent('OnNodePreExecute', THIS^);
END_METHOD

METHOD PRIVATE RegisterForPreExecuteEvent
VAR_INPUT
END_VAR
IF parentAsPreCheckedNode = 0 THEN
	RETURN;
END_IF

parentAsPreCheckedNode.OnEvent('OnNodePreExecute', this^);
END_METHOD

METHOD PUBLIC HandleEvent
VAR_INPUT
	Event : I_Event;
END_VAR
VAR
	nodePreExecuteEvent : I_NodePreExecuteEvent;
	preExecutionChecks : PreExecutionChecks;
END_VAR
IF NOT enable.Value THEN
	IF preExecutionCheckFailedAlarm.Active THEN
		preExecutionCheckFailedAlarm.Clear();
	END_IF
	RETURN;
END_IF

IF NOT __QUERYINTERFACE(Event, nodePreExecuteEvent) THEN
	RETURN;
END_IF

parentAsPreCheckedNode.PreExecutionCheck(preExecutionChecks);
IF preExecutionChecks.Failed THEN
	preExecutionCheckFailedAlarm.Raise(preExecutionChecks.Reason);
	nodePreExecuteEvent.Cancel();
	RETURN;
END_IF

preExecutionCheckFailedAlarm.Clear();
END_METHOD

END_FUNCTION_BLOCK

// IecDatatypesPack/IecDatatypesPack
{attribute 'linkalways'} 
{attribute 'no_explicit_call' := 'This FB is a CLASS and must be accessed using methods or properties'}
{attribute 'enable_dynamic_creation'}
FUNCTION_BLOCK IecDatatypesPack IMPLEMENTS I_GraphPack
VAR
	// _bit not included as this can only be part of a structure
	_bool : _BOOL(FALSE);
	_byte : _BYTE(0);
	_dint : _DINT(0);
	_dt : _DT(DT#1970-1-1-0:0:0);
	_dword : _DWORD(0);
	_int : _INT(0);
	_lint : _LINT(0);
	_lreal : _LREAL(0);
	_lword : _LWORD(0);
	_real : _REAL(0);
	_sint : _SINT(0);
	_time_of_day : _TIME_OF_DAY(TOD#0:0:0);
	_tod : _TOD(TOD#0:0:0);
	_udint : _UDINT(0);
	_uint : _UINT(0);
	_ulint : _ULINT(0);
	_usint : _USINT(0);
	_word : _WORD(0);
    _string : _STRING('');
END_VAR

METHOD RegisterWithDatatypes
VAR_INPUT
	Datatypes : I_Datatypes;
END_VAR
Datatypes.RegisterDatatype(_bool);
Datatypes.RegisterDatatype(_byte);
Datatypes.RegisterDatatype(_dint);
Datatypes.RegisterDatatype(_dt);
Datatypes.RegisterDatatype(_dword);
Datatypes.RegisterDatatype(_int);
Datatypes.RegisterDatatype(_lint);
Datatypes.RegisterDatatype(_lreal);
Datatypes.RegisterDatatype(_lword);
Datatypes.RegisterDatatype(_real);
Datatypes.RegisterDatatype(_sint);
Datatypes.RegisterDatatype(_time_of_day);
Datatypes.RegisterDatatype(_tod);
Datatypes.RegisterDatatype(_udint);
Datatypes.RegisterDatatype(_uint);
Datatypes.RegisterDatatype(_ulint);
Datatypes.RegisterDatatype(_usint);
Datatypes.RegisterDatatype(_word);
Datatypes.RegisterDatatype(_string);
END_METHOD

METHOD PUBLIC RegisterWithNodeFactory
VAR_INPUT
	NodeFactory : I_NodeFactory;
END_VAR
// not implemented
END_METHOD

END_FUNCTION_BLOCK
